//-- Priority -4
VA12: A     #o_ST_LSZ_Emptying; //Reporting on Time base
      A     #s_HLC_Report_Time_Active;
      O(    ;
      A     #o_ST_LSZ_Emptying; //Reporting on Status change
      FP    #s_FP_LSZ_Emptying;
      )     ;
      JCN   VA13;
      L     2; //Reporting "EMPTYING" Flushing
      T     #t_Segment_State;
      JU    VA20;

//-- Priority -5
VA13: A     #o_ST_Operational_On; //Reporting on Time base
      AN    #o_ST_LSZ_Full;
      AN    #o_ST_LSZ_Emptying;
      A     #s_HLC_Report_Time_Active;
      O(    ;
      A     #o_ST_Operational_On; //Reporting on Status change
      AN    #o_ST_LSZ_Full;
      AN    #o_ST_LSZ_Emptying;
      FP    #s_FP_Operation_On;
      )     ;
      JCN   VA99;
      L     1; //Reporting "OPERATIONAL" Ready to recieve the Bag
      T     #t_Segment_State;
      JU    VA20;

VA20: A     #s_HLC_Report_Time_Active; //IF HLC time interval expires
      O(    ; //OR
      L     #t_Segment_State; //Present Segment state
      L     #s_Prev_Segment_State; //Last report segment state
      <>I   ; //NOT-EQUAL  Report the Segment state to the DB-Event
      )     ;
      JCN   VA99;

//------------HLC REPORTING-------------//
      CALL "FC_Write_Event" (//Report the Segment state to the DB_Event
           i_Message_ID             := 1404,
           i_Event_value            := #t_Segment_State,
           i_DB_Event_Num           := #t_DB_Event_Num,
           o_Return_Value           := #t_Return_Value);


      L     #t_Segment_State;
      T     #s_Prev_Segment_State;

      CLR   ;
      =     #s_HLC_Report_Time_Active;

VA99: NOP   0;

      L     #t_Segment_State;
      L     #s_Prev_Segment_State;


END_FUNCTION_BLOCK

